(* PLC project static_torsion.project, CODESYS CODESYS V3.5 SP17 Patch 3 *)
(* stored: creationDateTime 1970-01-01T00:00:00, modificationDateTime 2026-06-22T15:12:39.4699931 *)

TYPE S_CTRL : STRUCT
  PowerOn : BIT;  (* Флаг включения регулятора сервопривода *)
  cmd_bit0 : BIT;  (* Команда управления работой стенда (3 бита) *)
  cmd_bit1 : BIT;  (* 000 = HALT; 001=JogCW; 010=JogCCW; 011=TORQUE_HOLD; 100=MOVE_TO_ANGLE *)
  cmd_bit2 : BIT;
  ResetTorque : BIT;  (* Обнуление момента *)
  ResetAngle : BIT;  (* Обнуление угла *)
  WriteRetain : BIT;  (* Запись уставок в память ПЛК *)
  ResetError : BIT;  (* Сброс ошибки привода *)
  ResetAlarm : BIT;  (* Сброс общей аварии стенда *)
  b9 : BIT;
  b10 : BIT;
  b11 : BIT;
  b12 : BIT;
  CalibrationMode : BIT;  (* Режим калибровки датчика момента *)
  b14 : BIT;
  ServiceMode : BIT;  (* Сервисный режим (прямое управление) *)
END_STRUCT;
END_TYPE
